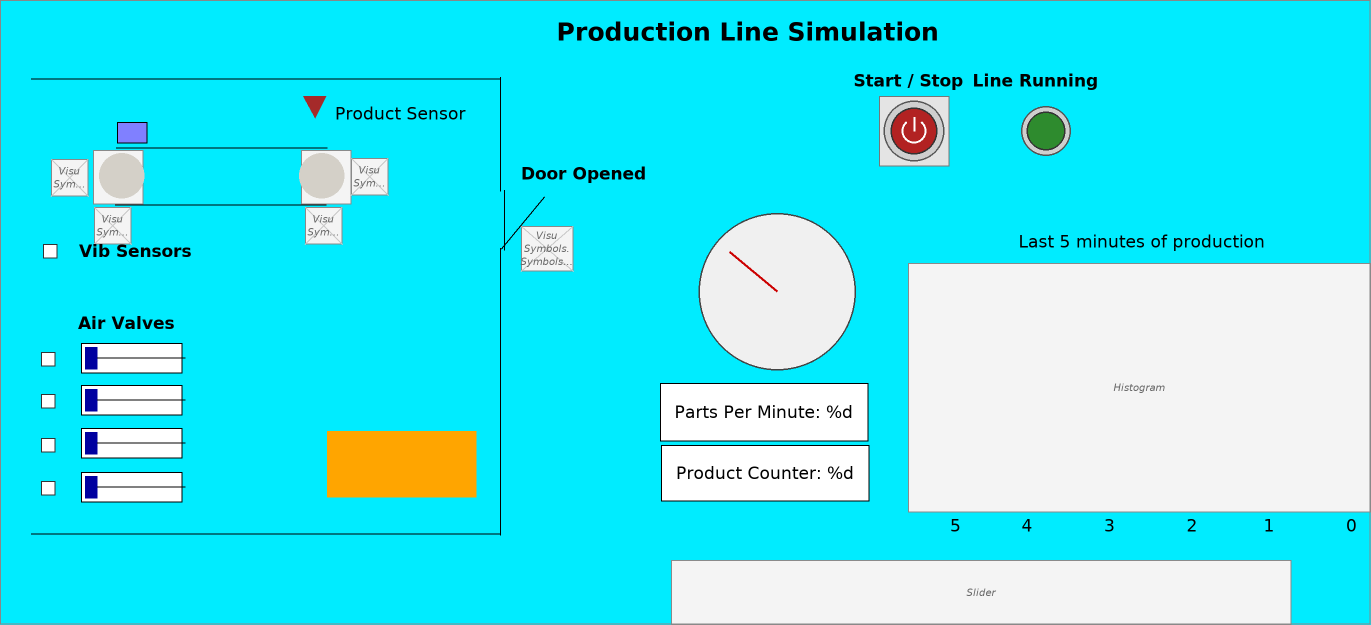
VISUALIZATION Visualization1  // 1371x625
    Pie (93,150 50x54), colour toggle: GVL_Visu.LineRunning
    Line (326,205) (115,205), colour toggle: GVL_Visu.LineRunning
    Line (327,148) (116,148), colour toggle: GVL_Visu.LineRunning
    Pie (301,150 50x54), colour toggle: GVL_Visu.LineRunning
    Meter360 (688,213 178x157), value: GVL_Visu.OkPartsPerMinRate, style: Meter-Meter360-Yellow, scale format: %.1f, scale 0..60
    Lamp1 (1010,102 72x58), variable: GVL_Visu.LineRunning, style: Lamp-Lamp1-Green
    Checkbox (39,344 33x30), variable: GVL_Visu.AirValveEnable[1]
    Line (500,77) (500,191)
    Line (500,248) (500,535)
    Line (500,534) (31,534)
    Line (544,197) (501,249), invisible if: NOT GVL_Visu.AutoMode
    Label (554,9 388x45), "Production Line Simulation"
    Image (521,226 52x45), colour toggle: GVL_Visu.LineRunning, invisible if: NOT GVL_Visu.AutoMode, image: VisuSymbols.Symbols.User
    RoundedRectangle (117,122 30x21)
        p3560616238: GVL_Visu.ProductPosition
    Rectangle (81,343 101x30)
    Group (85,347 100x22)
        p3560616238: GVL_Visu.AirValvePositionSim[1]
        Rectangle (0,0 12x22)
        Line (100,11) (12,11)
    Rectangle (81,385 101x30)
    Group (85,389 100x22)
        p3560616238: GVL_Visu.AirValvePositionSim[2]
        Rectangle (0,0 12x22)
        Line (100,11) (12,11)
    Rectangle (81,428 101x30)
    Group (85,432 100x22)
        p3560616238: GVL_Visu.AirValvePositionSim[3]
        Rectangle (0,0 12x22)
        Line (100,11) (12,11)
    Rectangle (81,472 101x30)
    Group (85,476 100x22)
        p3560616238: GVL_Visu.AirValvePositionSim[4]
        Rectangle (0,0 12x22)
        Line (100,11) (12,11)
    Line (500,79) (31,79)
    PowerSwitch (879,96 70x70), variable: GVL_Visu.ButtonStart, behaviour: TOGGLE, style: Switch-PowerSwitch-Red
    Rectangle (327,431 149x66), colour toggle: GVL_Visu.AutoMode, text list: 'TextList1', text index: GVL_Visu.AutoMode
    Ellipse (99,153 45x45), colour toggle: GVL_Visu.LineRunning
    Slider (671,560 620x65), variable: GVL_Visu.LineSpeed, scale 0..100
    Checkbox (39,386 34x30), variable: GVL_Visu.AirValveEnable[2]
    Checkbox (39,430 34x30), variable: GVL_Visu.AirValveEnable[3]
    Checkbox (39,473 34x30), variable: GVL_Visu.AirValveEnable[4]
    Ellipse (299,153 45x45), colour toggle: GVL_Visu.LineRunning
    Label (513,151 141x45), "Door Opened", invisible if: NOT GVL_Visu.AutoMode
    Polygon (303,96) (315,118) (326,96), colour toggle: GVL_Visu.SensorProductActive
    Label (330,91 141x45), "Product Sensor"
    Label (965,58 141x45), "Line Running"
    Line (504,190) (504,250), invisible if: GVL_Visu.AutoMode
    Label (56,306 141x34), "Air Valves"
    Image (51,159 37x37), angle 90, image: VisuSymbols.Symbols.Marker
    Image (94,207 37x37), image: VisuSymbols.Symbols.Marker
    Image (305,207 37x37), image: VisuSymbols.Symbols.Marker
    Image (351,158 37x37), angle -90, image: VisuSymbols.Symbols.Marker
    Label (65,234 141x34), "Vib Sensors"
    Histogram (908,263 463x249), scale format: %d, scale 0..60
        p1518820177: GVL_Visu.OkPartsPerMinHistorical
        p102497268: GVL_Visu.OkPartsPerMinHistorical
        p788070771: ARRAY [1..5] OF INT
    RoundedRectangle (661,445 208x56), "Product Counter: %d", text variable: GVL_Visu.OkProductCount
    RoundedRectangle (660,383 208x58), "Parts Per Minute: %d", text variable: GVL_Visu.OkPartsPerMinRate
    Label (997,219 290x45), "Last 5 minutes of production"
    Label (947,506 411x39), "5 4 3 2 1 0"
    Checkbox (41,236 33x30), variable: GVL_Visu.VibrationSensorsEnable
    Label (838,58 141x45), "Start / Stop"
END_VISUALIZATION

(* stored: Version 1.1.0.1, ProductVersion 3.1.4024.15
   Visu Visualization1: Id {7e5ded47-314c-404a-b2c3-829ddcb954e9} *)
